Staubli VAL3: remGetMaxA.pgx

program remGetMaxA(string& sReturn[] (dimensions=1))
  local string sCmd
begin
  // Return maximum allowed acceleration % for remote moves.
  //
  logMsg("call remGetMaxA")
  sCmd="GETMAXA"
  call remGetnGlobal(nMaxAccel,sCmd,sReturn)
end
